// TIA Portal V16 export
// export: Created 2021-11-12T13:33:13.0721327Z, ExportSetting WithDefaults, DisplayName Totally Integrated Automation Portal, DisplayVersion V16 Update 3, DisplayName TIA Portal Version Control Interface, DisplayVersion V16 Update 2, DisplayName TIA Portal Openness, DisplayVersion V16 Update 3, DisplayName SINAMICS Startdrive Advanced, DisplayVersion V16 Update 5, DisplayName SINAMICS Startdrive G130, G150, S120, S150, SINAMICS MV, S210, DisplayVersion V16 Update 5, DisplayName SINAMICS Startdrive G110M, G120, G120C, G120D, G120P, G115D, DisplayVersion V16 Update 5, DisplayName STEP 7 Professional, DisplayVersion V16 Update 3, DisplayName STEP 7 Safety, DisplayVersion V16, DisplayName WinCC UA Professional, DisplayVersion V16 Update 3
DATA_BLOCK "HMI_PARAM_400+UH11"   // DB150
{ S7_Optimized_Access := 'TRUE' }
VERSION : 0.1
// stored: AutoNumber true, DBAccessibleFromOPCUA true, IsOnlyStoredInLoadMemory false, IsRetainMemResEnabled false, IsWriteProtectedInAS false, MemoryReserve 100
   VAR
      xxxxx___BinarySensors___xxxxx : Byte;
      xxxxx___BinaryOthers___xxxxx : Byte;
      SF02_14 { S7_SetPoint := 'True'} : "UDT_CH_DI_Parameter";   // Automat start
      SF03_14 { S7_SetPoint := 'True'} : "UDT_CH_DI_Parameter";   // Error ack.
      SF04_14 { S7_SetPoint := 'True'} : "UDT_CH_DI_Parameter";   // Reset safety
      SF05_22 { S7_SetPoint := 'True'} : "UDT_CH_DI_Parameter";   // BSN4 chain blocking
      SF06_22 { S7_SetPoint := 'True'} : "UDT_CH_DI_Parameter";   // BSN5 chain blocking
      xxxxx___AnalogueSensors___xxxxx : Byte;
      xxxxx___Drives___xxxxx : Byte;
      xxxxx___Other___xxxxx : Byte;
      xxxxx___Alarms___xxxxx : Byte;
      ES { S7_SetPoint := 'True'} : "UDT_DI_Mon_Parameter";   // E-stop
      KF31 : "UDT_DI_Mon_Parameter";   // module KF31
   END_VAR
BEGIN
END_DATA_BLOCK
